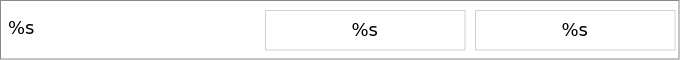
VISUALIZATION SingleRecipesParameterTypeString_1  // 680x60
VAR_IN_OUT
	stRecipeParameter : ST_VisuCtrlRecipeParameter;
END_VAR
    Textfield (265,10 200x40), "%s", text variable: stRecipeParameter.sValue
        OnMouseClick: write the text variable via VisuDialogs.Keypad
    Textfield (475,10 200x40), "%s", text variable: stRecipeParameter.sFileValue
    Textfield (5,8 250x40), "%s", text variable: stRecipeParameter.sName
END_VISUALIZATION

(* stored: Version 1.1.0.1, ProductVersion 3.1.4024.12
   Visu SingleRecipesParameterTypeString_1: Id {a772018d-8fd6-4b13-85bb-fa9dd2da89e9} *)
